FUNCTION_BLOCK TL_View (* Normal Traffic Light *)
  (* Standard: 61499-1; Classification: HMI; Function: Output; Type: 4xLED *)
  (* Version 0.4, 2018-07-27, JHC, Holobloc Inc, Updated I/O documentation. *)
  (* Version 0.3, 2011-03-28, JHC, Holobloc Inc, Updated documentation. *)
  (* Version 0.2, 2008-11-10, JHC, Holobloc Inc, Moved to fb.rt.doc. *)
  (* Version 0.1, 2008-06-04, JHC, Holobloc Inc, Updated DOCTYPE. *)
  (* Version 0.0, 2001-02-21, JHC, Rockwell Automation *)
  (* Compiler header: package fb.rt.template; import fb.rt.hmi.*; *)
  (* Compiler Java Sun JDK 1.7.0 *)
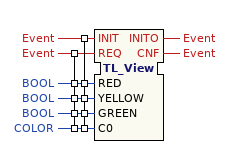
  EVENT_INPUT
    INIT WITH RED, YELLOW, GREEN, C0; (* Initialize *)
    REQ WITH RED, YELLOW, GREEN, C0; (* LED State/Color Update *)
  END_EVENT
  EVENT_OUTPUT
    INITO; (* INIT Confirm *)
    CNF; (* REQ Confirmation *)
  END_EVENT
  VAR_INPUT
    RED : BOOL; (* MSB - Most Significant Bit *)
    YELLOW : BOOL;
    GREEN : BOOL;
    C0 : COLOR := COLOR#white; (* OFF color *)
  END_VAR
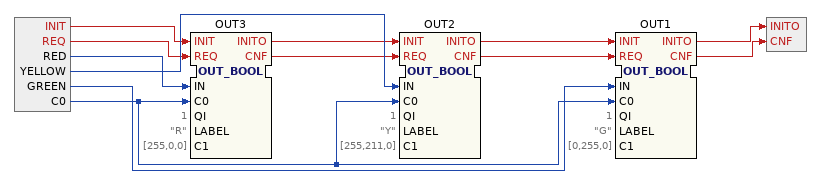
  FBS
    OUT3 : OUT_BOOL(QI := 1, LABEL := "R", C1 := [255,0,0]);
    OUT2 : OUT_BOOL(QI := 1, LABEL := "Y", C1 := [255,211,0]);
    OUT1 : OUT_BOOL(QI := 1, LABEL := "G", C1 := [0,255,0]);
  END_FBS
  EVENT_CONNECTIONS
    INIT TO OUT3.INIT;
    OUT3.INITO TO OUT2.INIT;
    OUT2.INITO TO OUT1.INIT;
    REQ TO OUT3.REQ;
    OUT3.CNF TO OUT2.REQ;
    OUT2.CNF TO OUT1.REQ;
    INIT TO OUT3.INIT;
    OUT3.INITO TO OUT2.INIT;
    OUT2.INITO TO OUT1.INIT;
    REQ TO OUT3.REQ;
    OUT3.CNF TO OUT2.REQ;
    OUT2.CNF TO OUT1.REQ;
    OUT1.INITO TO INITO;
    OUT1.CNF TO CNF;
  END_CONNECTIONS
  DATA_CONNECTIONS
    RED TO OUT3.IN;
    YELLOW TO OUT2.IN;
    GREEN TO OUT1.IN;
    C0 TO OUT3.C0;
    C0 TO OUT2.C0;
    C0 TO OUT1.C0;
    RED TO OUT3.IN;
    YELLOW TO OUT2.IN;
    GREEN TO OUT1.IN;
    C0 TO OUT3.C0;
    C0 TO OUT2.C0;
    C0 TO OUT1.C0;
  END_CONNECTIONS
END_FUNCTION_BLOCK
